PROGRAM MAIN
VAR
Elevation : FB_Elevation;
Azimuth : FB_Azimuth;
END_VAR

Elevation();
Azimuth();

END_PROGRAM

(* stored: Version 1.1.0.1, ProductVersion 3.1.4024.15
   POU MAIN: Id {c126dce8-c39b-4cfd-9642-3394e5392cc2}, SpecialFunc None *)
